PROGRAM Axe_05_Z_Laser
VAR	
	ZLaser: FB_axe_ZLaser;
	RE_palpage_ok: R_TRIG;
	Asserv_Torche_On_test: BOOL;
	TON_Decoupe_recente		:TON;	
	FE_Decoupe_en_cours		:F_TRIG;
	TON_decoupe_manu: TON;
	TP_not_machine_en_service: TP;
	A_completer: BOOL;
	TestKerf: BOOL;
	Reset_Z: BOOL;
	TOF_DecMan	:TOF;
	EXemple: LREAL;
END_VAR

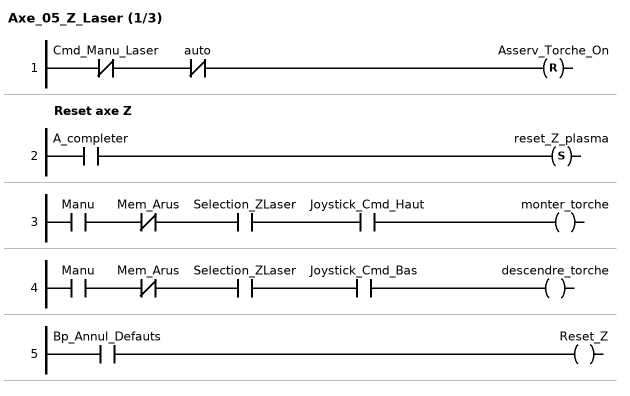
// NETWORK 1
Asserv_Torche_On R= NOT Cmd_Manu_Laser AND NOT auto;

// NETWORK 2: Reset axe Z
reset_Z_plasma S= A_completer;

// NETWORK 3
monter_torche := Manu AND NOT Mem_Arus AND Selection_ZLaser AND Joystick_Cmd_Haut;

// NETWORK 4
descendre_torche := Manu AND NOT Mem_Arus AND Selection_ZLaser AND Joystick_Cmd_Bas;

// NETWORK 5
Reset_Z := Bp_Annul_Defauts;

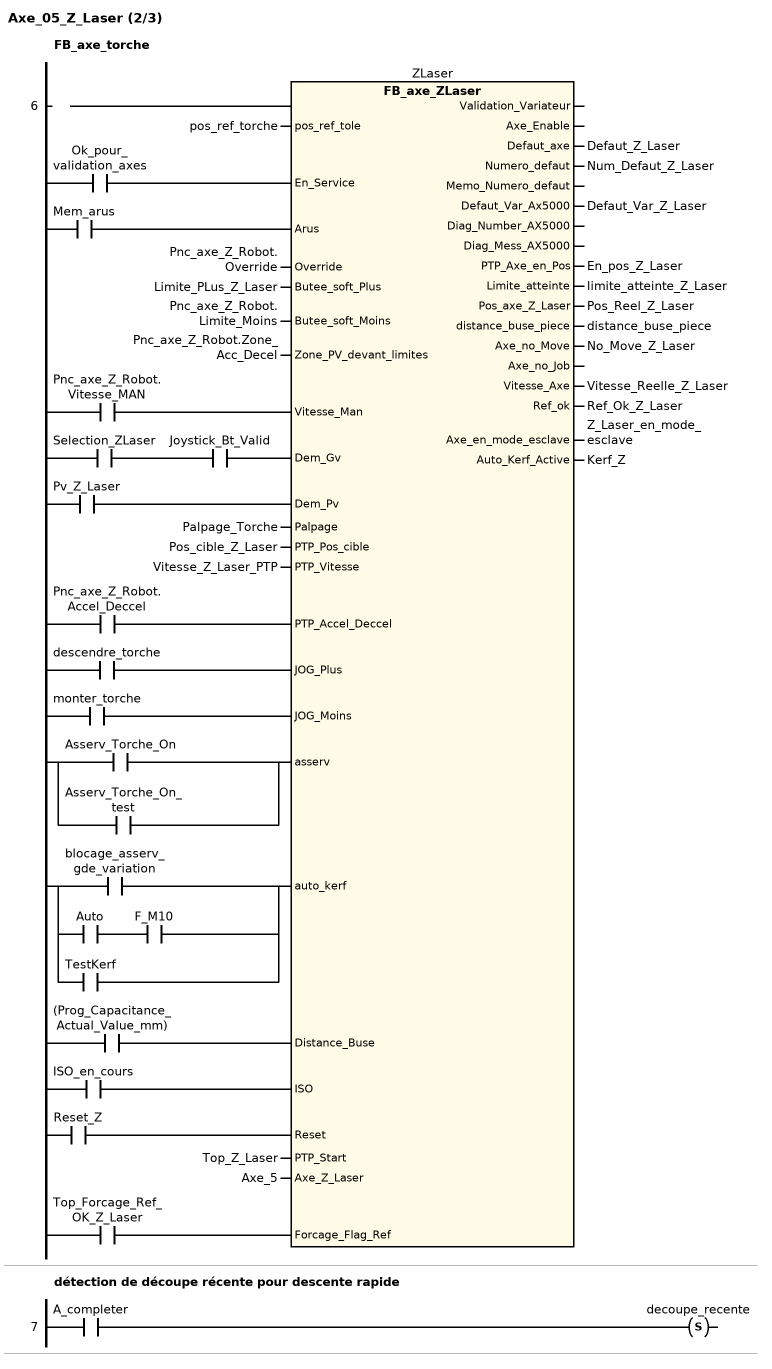
// NETWORK 6: FB_axe_torche
ZLaser(
    pos_ref_tole := pos_ref_torche,
    En_Service := Ok_pour_validation_axes,
    Arus := Mem_arus,
    Override := Pnc_axe_Z_Robot.Override,
    Butee_soft_Plus := Limite_PLus_Z_Laser,
    Butee_soft_Moins := Pnc_axe_Z_Robot.Limite_Moins,
    Zone_PV_devant_limites := Pnc_axe_Z_Robot.Zone_Acc_Decel,
    Vitesse_Man := Pnc_axe_Z_Robot.Vitesse_MAN,
    Dem_Gv := Selection_ZLaser AND Joystick_Bt_Valid,
    Dem_Pv := Pv_Z_Laser,
    Palpage := Palpage_Torche,
    PTP_Pos_cible := Pos_cible_Z_Laser,
    PTP_Vitesse := Vitesse_Z_Laser_PTP,
    PTP_Accel_Deccel := Pnc_axe_Z_Robot.Accel_Deccel,
    JOG_Plus := descendre_torche,
    JOG_Moins := monter_torche,
    asserv := Asserv_Torche_On OR Asserv_Torche_On_test,
    auto_kerf := blocage_asserv_gde_variation OR Auto AND F_M10 OR TestKerf,
    Distance_Buse := (Prog_Capacitance_Actual_Value_mm),
    ISO := ISO_en_cours,
    Reset := Reset_Z,
    PTP_Start := Top_Z_Laser,
    Axe_Z_Laser := Axe_5,
    Forcage_Flag_Ref := Top_Forcage_Ref_OK_Z_Laser,
    Defaut_axe => Defaut_Z_Laser,
    Numero_defaut => Num_Defaut_Z_Laser,
    Defaut_Var_Ax5000 => Defaut_Var_Z_Laser,
    PTP_Axe_en_Pos => En_pos_Z_Laser,
    Limite_atteinte => limite_atteinte_Z_Laser,
    Pos_axe_Z_Laser => Pos_Reel_Z_Laser,
    distance_buse_piece => distance_buse_piece,
    Axe_no_Move => No_Move_Z_Laser,
    Vitesse_Axe => Vitesse_Reelle_Z_Laser,
    Ref_ok => Ref_Ok_Z_Laser,
    Axe_en_mode_esclave => Z_Laser_en_mode_esclave,
    Auto_Kerf_Active => Kerf_Z); // FB_axe_ZLaser

// NETWORK 7: détection de découpe récente pour descente rapide
decoupe_recente S= A_completer;

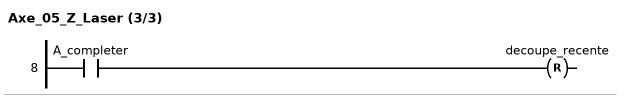
// NETWORK 8
decoupe_recente R= A_completer;

END_PROGRAM

(* stored: Version 1.1.0.1
   POU Axe_05_Z_Laser: Id {8b3232da-870b-493c-8747-341602195cf2}, SpecialFunc None *)
